// TIA Portal project "babu_3wayTrafficLight" (V15)

(* hardware
DEVICE "S7-1200 station_1"  S7-1200 Station
   slot 0: "Rack_0"  S7-1200 Rack  Rack  V1.0
   slot 1: "PLC_1"  CPU 1212C DC/DC/DC  6ES7 212-1AE40-0XB0  V4.2
*)

// ===== PLC "PLC_1"  CPU 1212C DC/DC/DC =====

VAR_GLOBAL   // PLC tag table "Default tag table"
   "PUSH BUTTON" AT %I0.0 : Bool;
   "PUSH BUTTON MEMORY" AT %M0.1 : Bool;
   "INITIALIZE" AT %M0.2 : Bool;
   "R1M" AT %M0.3 : Bool;
   "R2M" AT %M0.4 : Bool;
   "G3M" AT %M0.5 : Bool;
   "Y1M" AT %M0.6 : Bool;
   "G1M" AT %M0.7 : Bool;
   "R3M" AT %M1.0 : Bool;
   "Y2M" AT %M1.1 : Bool;
   "G2M" AT %M1.2 : Bool;
   "Y3M" AT %M1.3 : Bool;
   "SEQ1" AT %M0.0 : Bool;
   "SEQ2" AT %M1.4 : Bool;
   "SEQ3" AT %M1.5 : Bool;
   "SEQ4" AT %M1.6 : Bool;
   "SEQ5" AT %M1.7 : Bool;
   "SEQ6" AT %M2.0 : Bool;
   "ERROR" AT %M2.1 : Bool;
END_VAR

VAR_GLOBAL   // PLC tag table "Tag table_1"
   "R1" AT %Q0.7 : Bool;
   "R3" AT %Q1.0 : Bool;
   "R2" AT %Q0.3 : Bool;
   "Y1" AT %Q0.1 : Bool;
   "Y2" AT %Q0.4 : Bool;
   "Y3" AT %Q0.6 : Bool;
   "G1" AT %Q0.2 : Bool;
   "G2" AT %Q0.5 : Bool;
   "G3" AT %Q0.0 : Bool;
END_VAR

// folder: System blocks/Program resources

DATA_BLOCK "IEC_Timer_0_DB"   // DB1
{ S7_Optimized_Access := 'TRUE' }
AUTHOR : Simatic
FAMILY : IEC
NAME : IEC_TMR
VERSION : 1.0
// stored: InstanceOfName IEC_TIMER
"IEC_TIMER"
BEGIN
END_DATA_BLOCK

DATA_BLOCK "IEC_Timer_0_DB_1"   // DB2
{ S7_Optimized_Access := 'TRUE' }
AUTHOR : Simatic
FAMILY : IEC
NAME : IEC_TMR
VERSION : 1.0
// stored: InstanceOfName IEC_TIMER
"IEC_TIMER"
BEGIN
END_DATA_BLOCK

DATA_BLOCK "IEC_Timer_0_DB_2"   // DB3
{ S7_Optimized_Access := 'TRUE' }
AUTHOR : Simatic
FAMILY : IEC
NAME : IEC_TMR
VERSION : 1.0
// stored: InstanceOfName IEC_TIMER
"IEC_TIMER"
BEGIN
END_DATA_BLOCK

DATA_BLOCK "IEC_Timer_0_DB_3"   // DB4
{ S7_Optimized_Access := 'TRUE' }
AUTHOR : Simatic
FAMILY : IEC
NAME : IEC_TMR
VERSION : 1.0
// stored: InstanceOfName IEC_TIMER
"IEC_TIMER"
BEGIN
END_DATA_BLOCK

DATA_BLOCK "IEC_Timer_0_DB_4"   // DB5
{ S7_Optimized_Access := 'TRUE' }
AUTHOR : Simatic
FAMILY : IEC
NAME : IEC_TMR
VERSION : 1.0
// stored: InstanceOfName IEC_TIMER
"IEC_TIMER"
BEGIN
END_DATA_BLOCK

DATA_BLOCK "IEC_Timer_0_DB_5"   // DB6
{ S7_Optimized_Access := 'TRUE' }
AUTHOR : Simatic
FAMILY : IEC
NAME : IEC_TMR
VERSION : 1.0
// stored: InstanceOfName IEC_TIMER
"IEC_TIMER"
BEGIN
END_DATA_BLOCK

DATA_BLOCK "IEC_Timer_0_DB_6"   // DB7
{ S7_Optimized_Access := 'TRUE' }
AUTHOR : Simatic
FAMILY : IEC
NAME : IEC_TMR
VERSION : 1.0
// stored: InstanceOfName IEC_TIMER
"IEC_TIMER"
BEGIN
END_DATA_BLOCK

DATA_BLOCK "IEC_Timer_0_DB_7"   // DB8
{ S7_Optimized_Access := 'TRUE' }
AUTHOR : Simatic
FAMILY : IEC
NAME : IEC_TMR
VERSION : 1.0
// stored: InstanceOfName IEC_TIMER
"IEC_TIMER"
BEGIN
END_DATA_BLOCK

DATA_BLOCK "IEC_Timer_0_DB_8"   // DB9
{ S7_Optimized_Access := 'TRUE' }
AUTHOR : Simatic
FAMILY : IEC
NAME : IEC_TMR
VERSION : 1.0
// stored: InstanceOfName IEC_TIMER
"IEC_TIMER"
BEGIN
END_DATA_BLOCK

DATA_BLOCK "IEC_Timer_0_DB_9"   // DB10
{ S7_Optimized_Access := 'TRUE' }
AUTHOR : Simatic
FAMILY : IEC
NAME : IEC_TMR
VERSION : 1.0
// stored: InstanceOfName IEC_TIMER
"IEC_TIMER"
BEGIN
END_DATA_BLOCK

DATA_BLOCK "IEC_Timer_0_DB_10"   // DB11
{ S7_Optimized_Access := 'TRUE' }
AUTHOR : Simatic
FAMILY : IEC
NAME : IEC_TMR
VERSION : 1.0
// stored: InstanceOfName IEC_TIMER
"IEC_TIMER"
BEGIN
END_DATA_BLOCK

DATA_BLOCK "IEC_Timer_0_DB_11"   // DB12
{ S7_Optimized_Access := 'TRUE' }
AUTHOR : Simatic
FAMILY : IEC
NAME : IEC_TMR
VERSION : 1.0
// stored: InstanceOfName IEC_TIMER
"IEC_TIMER"
BEGIN
END_DATA_BLOCK

DATA_BLOCK "IEC_Timer_0_DB_12"   // DB13
{ S7_Optimized_Access := 'TRUE' }
AUTHOR : Simatic
FAMILY : IEC
NAME : IEC_TMR
VERSION : 1.0
// stored: InstanceOfName IEC_TIMER
"IEC_TIMER"
BEGIN
END_DATA_BLOCK

DATA_BLOCK "IEC_Timer_0_DB_13"   // DB14
{ S7_Optimized_Access := 'TRUE' }
AUTHOR : Simatic
FAMILY : IEC
NAME : IEC_TMR
VERSION : 1.0
// stored: InstanceOfName IEC_TIMER
"IEC_TIMER"
BEGIN
END_DATA_BLOCK

DATA_BLOCK "IEC_Timer_0_DB_14"   // DB15
{ S7_Optimized_Access := 'TRUE' }
AUTHOR : Simatic
FAMILY : IEC
NAME : IEC_TMR
VERSION : 1.0
// stored: InstanceOfName IEC_TIMER
"IEC_TIMER"
BEGIN
END_DATA_BLOCK

DATA_BLOCK "IEC_Timer_0_DB_15"   // DB16
{ S7_Optimized_Access := 'TRUE' }
AUTHOR : Simatic
FAMILY : IEC
NAME : IEC_TMR
VERSION : 1.0
// stored: InstanceOfName IEC_TIMER
"IEC_TIMER"
BEGIN
END_DATA_BLOCK

DATA_BLOCK "IEC_Timer_0_DB_17"   // DB18
{ S7_Optimized_Access := 'TRUE' }
AUTHOR : Simatic
FAMILY : IEC
NAME : IEC_TMR
VERSION : 1.0
// stored: InstanceOfName IEC_TIMER
"IEC_TIMER"
BEGIN
END_DATA_BLOCK

DATA_BLOCK "IEC_Timer_0_DB_18"   // DB19
{ S7_Optimized_Access := 'TRUE' }
AUTHOR : Simatic
FAMILY : IEC
NAME : IEC_TMR
VERSION : 1.0
// stored: InstanceOfName IEC_TIMER
"IEC_TIMER"
BEGIN
END_DATA_BLOCK

DATA_BLOCK "IEC_Timer_0_DB_19"   // DB20
{ S7_Optimized_Access := 'TRUE' }
AUTHOR : Simatic
FAMILY : IEC
NAME : IEC_TMR
VERSION : 1.0
// stored: InstanceOfName IEC_TIMER
"IEC_TIMER"
BEGIN
END_DATA_BLOCK

DATA_BLOCK "IEC_Timer_0_DB_20"   // DB21
{ S7_Optimized_Access := 'TRUE' }
AUTHOR : Simatic
FAMILY : IEC
NAME : IEC_TMR
VERSION : 1.0
// stored: InstanceOfName IEC_TIMER
"IEC_TIMER"
BEGIN
END_DATA_BLOCK

DATA_BLOCK "IEC_Timer_0_DB_21"   // DB22
{ S7_Optimized_Access := 'TRUE' }
AUTHOR : Simatic
FAMILY : IEC
NAME : IEC_TMR
VERSION : 1.0
// stored: InstanceOfName IEC_TIMER
"IEC_TIMER"
BEGIN
END_DATA_BLOCK

DATA_BLOCK "IEC_Timer_0_DB_22"   // DB23
{ S7_Optimized_Access := 'TRUE' }
AUTHOR : Simatic
FAMILY : IEC
NAME : IEC_TMR
VERSION : 1.0
// stored: InstanceOfName IEC_TIMER
"IEC_TIMER"
BEGIN
END_DATA_BLOCK

DATA_BLOCK "IEC_Timer_0_DB_23"   // DB24
{ S7_Optimized_Access := 'TRUE' }
AUTHOR : Simatic
FAMILY : IEC
NAME : IEC_TMR
VERSION : 1.0
// stored: InstanceOfName IEC_TIMER
"IEC_TIMER"
BEGIN
END_DATA_BLOCK

DATA_BLOCK "IEC_Timer_0_DB_25"   // DB26
{ S7_Optimized_Access := 'TRUE' }
AUTHOR : Simatic
FAMILY : IEC
NAME : IEC_TMR
VERSION : 1.0
// stored: InstanceOfName IEC_TIMER
"IEC_TIMER"
BEGIN
END_DATA_BLOCK

// folder: (top level)

ORGANIZATION_BLOCK "Main"   // OB1, LAD, ProgramCycle
TITLE = "Main Program Sweep (Cycle)"
{ S7_Optimized_Access := 'TRUE' }
VERSION : 0.1
   VAR_INPUT
      Initial_Call : Bool;   // Initial call of this OB
      Remanence : Bool;   // =True, if remanent data are available
   END_VAR
   VAR_TEMP   // added for the SCL form of the ladder/FBD networks
      _w1 : Bool;
      _w2 : Bool;
      _w3 : Bool;
   END_VAR
BEGIN

REGION Network 1
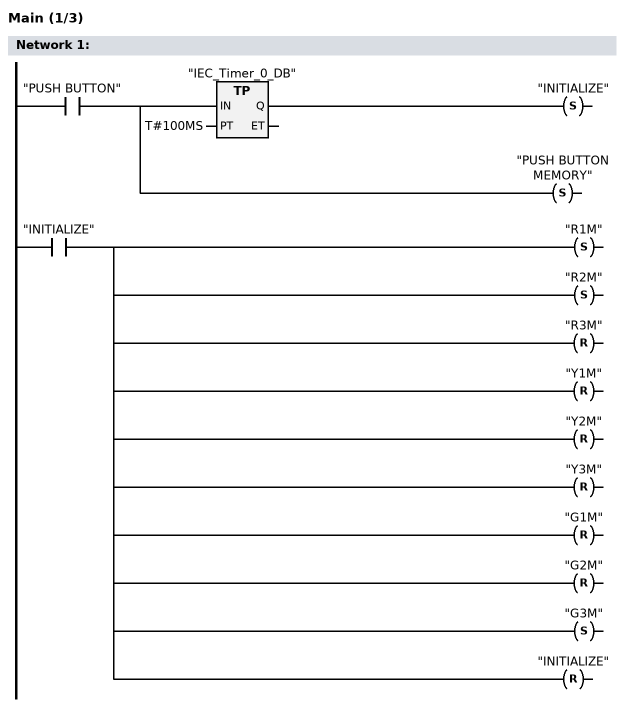
   "IEC_Timer_0_DB".TP(IN := "PUSH BUTTON", PT := T#100MS);
   IF "IEC_Timer_0_DB".Q THEN "INITIALIZE" := TRUE; END_IF;
   IF "PUSH BUTTON" THEN "PUSH BUTTON MEMORY" := TRUE; END_IF;
   IF "INITIALIZE" THEN
       "R1M" := TRUE;
       "R2M" := TRUE;
       "R3M" := FALSE;
       "Y1M" := FALSE;
       "Y2M" := FALSE;
       "Y3M" := FALSE;
       "G1M" := FALSE;
       "G2M" := FALSE;
       "G3M" := TRUE;
       "INITIALIZE" := FALSE;
   END_IF;
END_REGION

REGION Network 2
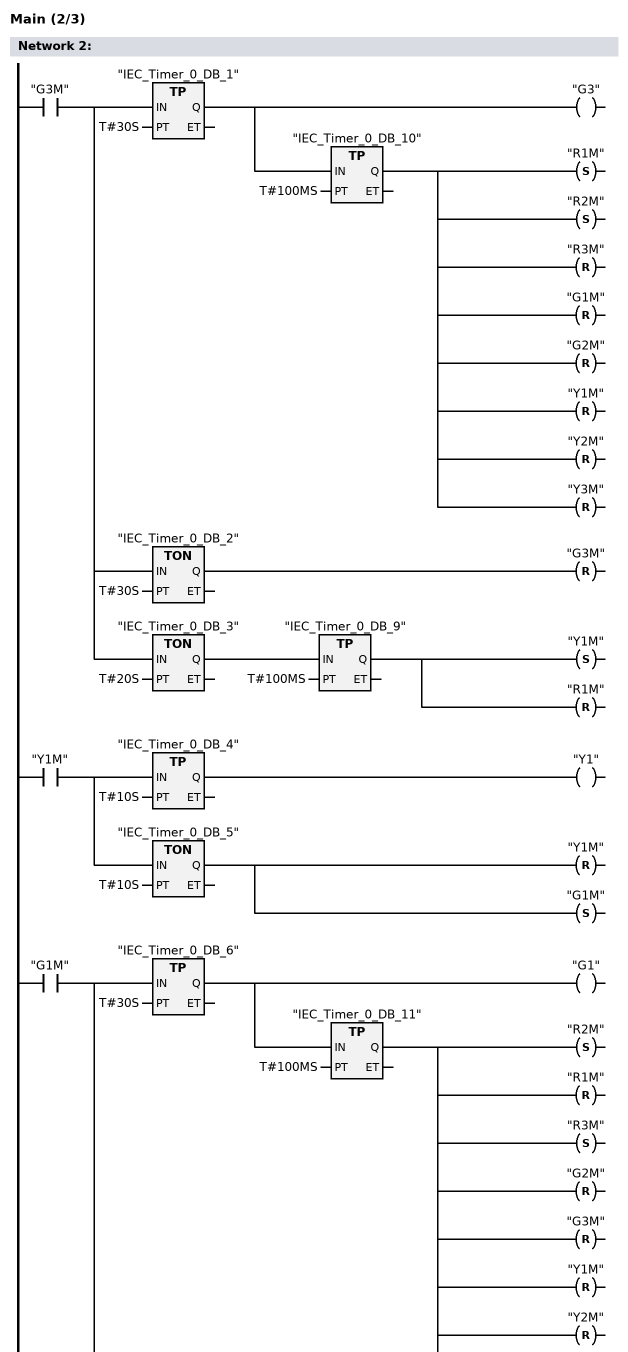
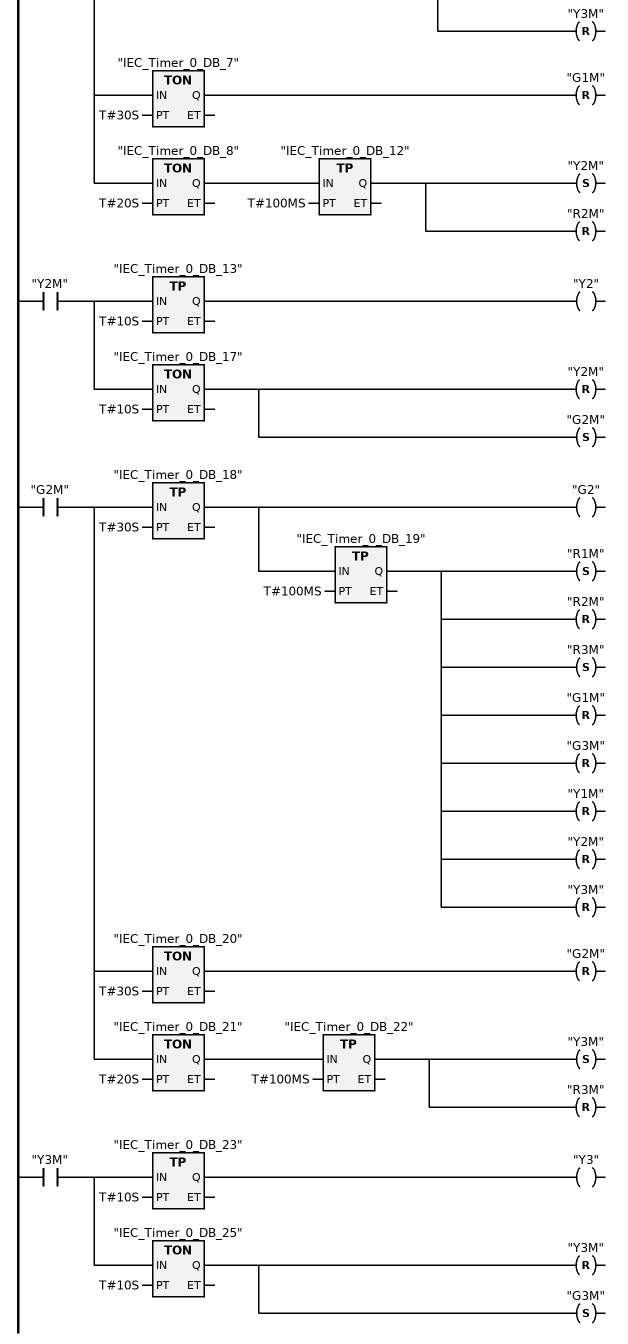
   "IEC_Timer_0_DB_1".TP(IN := "G3M", PT := T#30S);
   "G3" := "IEC_Timer_0_DB_1".Q;
   "IEC_Timer_0_DB_10".TP(IN := "IEC_Timer_0_DB_1".Q, PT := T#100MS);
   IF "IEC_Timer_0_DB_10".Q THEN
       "R1M" := TRUE;
       "R2M" := TRUE;
       "R3M" := FALSE;
       "G1M" := FALSE;
       "G2M" := FALSE;
       "Y1M" := FALSE;
       "Y2M" := FALSE;
       "Y3M" := FALSE;
   END_IF;
   "IEC_Timer_0_DB_2".TON(IN := "G3M", PT := T#30S);
   #_w1 := "G3M";
   IF "IEC_Timer_0_DB_2".Q THEN "G3M" := FALSE; END_IF;
   "IEC_Timer_0_DB_3".TON(IN := #_w1, PT := T#20S);
   "IEC_Timer_0_DB_9".TP(IN := "IEC_Timer_0_DB_3".Q, PT := T#100MS);
   IF "IEC_Timer_0_DB_9".Q THEN
       "Y1M" := TRUE;
       "R1M" := FALSE;
   END_IF;
   "IEC_Timer_0_DB_4".TP(IN := "Y1M", PT := T#10S);
   "Y1" := "IEC_Timer_0_DB_4".Q;
   "IEC_Timer_0_DB_5".TON(IN := "Y1M", PT := T#10S);
   IF "IEC_Timer_0_DB_5".Q THEN
       "Y1M" := FALSE;
       "G1M" := TRUE;
   END_IF;
   "IEC_Timer_0_DB_6".TP(IN := "G1M", PT := T#30S);
   "G1" := "IEC_Timer_0_DB_6".Q;
   "IEC_Timer_0_DB_11".TP(IN := "IEC_Timer_0_DB_6".Q, PT := T#100MS);
   IF "IEC_Timer_0_DB_11".Q THEN
       "R2M" := TRUE;
       "R1M" := FALSE;
       "R3M" := TRUE;
       "G2M" := FALSE;
       "G3M" := FALSE;
       "Y1M" := FALSE;
       "Y2M" := FALSE;
       "Y3M" := FALSE;
   END_IF;
   "IEC_Timer_0_DB_7".TON(IN := "G1M", PT := T#30S);
   #_w2 := "G1M";
   IF "IEC_Timer_0_DB_7".Q THEN "G1M" := FALSE; END_IF;
   "IEC_Timer_0_DB_8".TON(IN := #_w2, PT := T#20S);
   "IEC_Timer_0_DB_12".TP(IN := "IEC_Timer_0_DB_8".Q, PT := T#100MS);
   IF "IEC_Timer_0_DB_12".Q THEN
       "Y2M" := TRUE;
       "R2M" := FALSE;
   END_IF;
   "IEC_Timer_0_DB_13".TP(IN := "Y2M", PT := T#10S);
   "Y2" := "IEC_Timer_0_DB_13".Q;
   "IEC_Timer_0_DB_17".TON(IN := "Y2M", PT := T#10S);
   IF "IEC_Timer_0_DB_17".Q THEN
       "Y2M" := FALSE;
       "G2M" := TRUE;
   END_IF;
   "IEC_Timer_0_DB_18".TP(IN := "G2M", PT := T#30S);
   "G2" := "IEC_Timer_0_DB_18".Q;
   "IEC_Timer_0_DB_19".TP(IN := "IEC_Timer_0_DB_18".Q, PT := T#100MS);
   IF "IEC_Timer_0_DB_19".Q THEN
       "R1M" := TRUE;
       "R2M" := FALSE;
       "R3M" := TRUE;
       "G1M" := FALSE;
       "G3M" := FALSE;
       "Y1M" := FALSE;
       "Y2M" := FALSE;
       "Y3M" := FALSE;
   END_IF;
   "IEC_Timer_0_DB_20".TON(IN := "G2M", PT := T#30S);
   #_w3 := "G2M";
   IF "IEC_Timer_0_DB_20".Q THEN "G2M" := FALSE; END_IF;
   "IEC_Timer_0_DB_21".TON(IN := #_w3, PT := T#20S);
   "IEC_Timer_0_DB_22".TP(IN := "IEC_Timer_0_DB_21".Q, PT := T#100MS);
   IF "IEC_Timer_0_DB_22".Q THEN
       "Y3M" := TRUE;
       "R3M" := FALSE;
   END_IF;
   "IEC_Timer_0_DB_23".TP(IN := "Y3M", PT := T#10S);
   "Y3" := "IEC_Timer_0_DB_23".Q;
   "IEC_Timer_0_DB_25".TON(IN := "Y3M", PT := T#10S);
   IF "IEC_Timer_0_DB_25".Q THEN
       "Y3M" := FALSE;
       "G3M" := TRUE;
   END_IF;
END_REGION

REGION Network 3
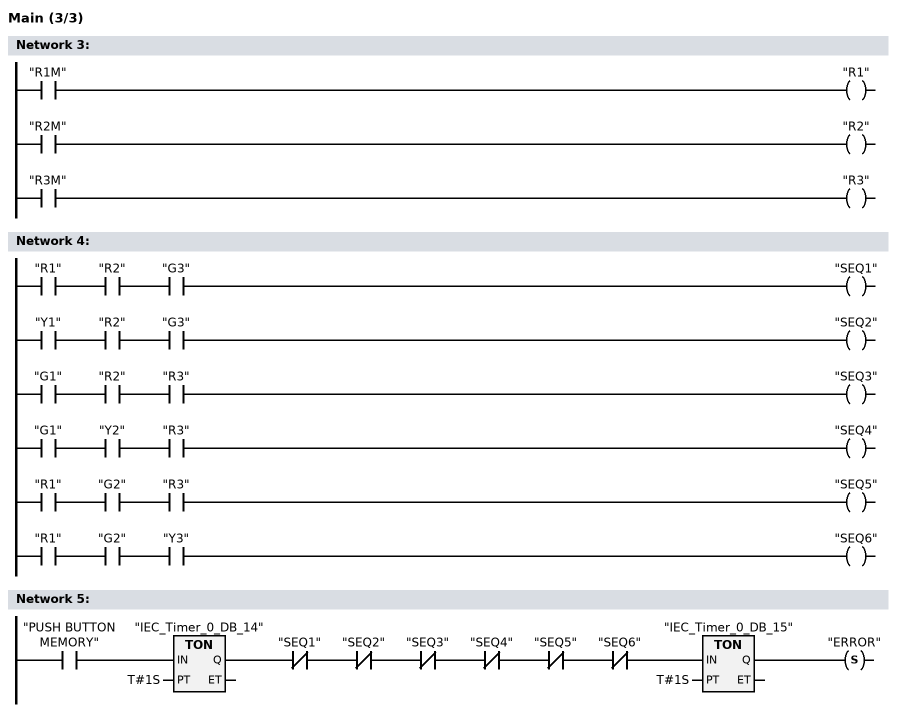
   RUNG wire#powerrail
      Contact( "R1M" )
      Coil( "R1" )
   END_RUNG
   RUNG wire#powerrail
      Contact( "R2M" )
      Coil( "R2" )
   END_RUNG
   RUNG wire#powerrail
      Contact( "R3M" )
      Coil( "R3" )
   END_RUNG
   // the same network as SCL:
   "R1" := "R1M";
   "R2" := "R2M";
   "R3" := "R3M";
END_REGION

REGION Network 4
   RUNG wire#powerrail
      Contact( "R1" )
      Contact( "R2" )
      Contact( "G3" )
      Coil( "SEQ1" )
   END_RUNG
   RUNG wire#powerrail
      Contact( "Y1" )
      Contact( "R2" )
      Contact( "G3" )
      Coil( "SEQ2" )
   END_RUNG
   RUNG wire#powerrail
      Contact( "G1" )
      Contact( "R2" )
      Contact( "R3" )
      Coil( "SEQ3" )
   END_RUNG
   RUNG wire#powerrail
      Contact( "G1" )
      Contact( "Y2" )
      Contact( "R3" )
      Coil( "SEQ4" )
   END_RUNG
   RUNG wire#powerrail
      Contact( "R1" )
      Contact( "G2" )
      Contact( "R3" )
      Coil( "SEQ5" )
   END_RUNG
   RUNG wire#powerrail
      Contact( "R1" )
      Contact( "G2" )
      Contact( "Y3" )
      Coil( "SEQ6" )
   END_RUNG
   // the same network as SCL:
   "SEQ1" := "R1" AND "R2" AND "G3";
   "SEQ2" := "Y1" AND "R2" AND "G3";
   "SEQ3" := "G1" AND "R2" AND "R3";
   "SEQ4" := "G1" AND "Y2" AND "R3";
   "SEQ5" := "R1" AND "G2" AND "R3";
   "SEQ6" := "R1" AND "G2" AND "Y3";
END_REGION

REGION Network 5
   "IEC_Timer_0_DB_14".TON(IN := "PUSH BUTTON MEMORY", PT := T#1S);
   "IEC_Timer_0_DB_15".TON(IN := "IEC_Timer_0_DB_14".Q AND NOT "SEQ1" AND NOT "SEQ2" AND NOT "SEQ3" AND NOT "SEQ4" AND NOT "SEQ5" AND NOT "SEQ6",
                           PT := T#1S);
   IF "IEC_Timer_0_DB_15".Q THEN "ERROR" := TRUE; END_IF;
END_REGION
END_ORGANIZATION_BLOCK